FUNCTION TFClearApprendimento : BOOL //Funzione che pulisce la struttura dell'apprendimento
VAR_INPUT
	Apprendimento : POINTER TO TFMachinePalletizer_CoordinateApprendimento;
END_VAR
VAR
	i : INT;
END_VAR

MEMSET(ADR(Apprendimento^),0,SIZEOF(Apprendimento^));
TFClearApprendimento := TRUE;

END_FUNCTION

(* stored: Version 1.1.0.1, ProductVersion 3.1.4024.11
   POU TFClearApprendimento: Id {0236d6ed-ea2f-4f43-a863-6e38fa18c1fb}, SpecialFunc None *)
